(* IEC 61131-3 sources: plc_generation_empirical_study/datasets/task_bank_c06_reverse_bounded_runtime_v0_3/tasks/C06_V04_lean_composite/negative_control, 1 file *)

(* ---- NC1.st ---- *)
FUNCTION_BLOCK C06_V04_lean_composite
VAR_INPUT
    A_Info : BOOL;
    A_Warning : BOOL;
    A_Trip : BOOL;
    A_Emergency : BOOL;
    A_Suppress : BOOL;
    B_AddItem : BOOL;
    B_RemoveItem : BOOL;
    B_Reset : BOOL;
    B_Capacity : INT;
    SubsystemBEnable : BOOL;
    CrossReset : BOOL;
END_VAR
VAR_OUTPUT
    A_Active : BOOL;
    A_Level : INT;
    B_Count : INT;
    B_Empty : BOOL;
    B_Full : BOOL;
    B_Conflict : BOOL;
    CrossReady : BOOL;
    CrossBlocked : BOOL;
END_VAR
VAR
    B_PrevAdd : BOOL := FALSE;
    B_PrevRemove : BOOL := FALSE;
END_VAR

IF A_Emergency THEN
    A_Level := 4;
    A_Active := TRUE;
ELSIF A_Suppress THEN
    A_Level := 0;
    A_Active := FALSE;
ELSIF A_Trip THEN
    A_Level := 3;
    A_Active := TRUE;
ELSIF A_Warning THEN
    A_Level := 2;
    A_Active := TRUE;
ELSIF A_Info THEN
    A_Level := 1;
    A_Active := TRUE;
ELSE
    A_Level := 0;
    A_Active := FALSE;
END_IF;

IF CrossReset THEN
    CrossReady := FALSE;
ELSIF A_Active THEN
    CrossReady := TRUE;
END_IF;
CrossBlocked := FALSE;

IF SubsystemBEnable AND CrossReady THEN
    B_Conflict := FALSE;
    IF B_Reset THEN
        B_Count := 0;
    ELSIF B_AddItem AND (NOT B_PrevAdd) AND B_RemoveItem AND (NOT B_PrevRemove) THEN
        B_Conflict := TRUE;
    ELSIF B_AddItem AND (NOT B_PrevAdd) AND (B_Count < B_Capacity) THEN
        B_Count := B_Count + 1;
    ELSIF B_RemoveItem AND (NOT B_PrevRemove) AND (B_Count > 0) THEN
        B_Count := B_Count - 1;
    END_IF;
    B_Empty := B_Count = 0;
    B_Full := B_Count >= B_Capacity;
    B_PrevAdd := B_AddItem;
    B_PrevRemove := B_RemoveItem;
ELSE
    B_Count := 0;
    B_Empty := FALSE;
    B_Full := FALSE;
    B_Conflict := FALSE;
END_IF;

END_FUNCTION_BLOCK
